// TIA Portal V20 export
TYPE "typeCmControlNodeInterlock"
// stored: Namespace Unit1.Em0
   STRUCT
      stacker1NgBoxLoading : "LER_typeTwoWayActuatorInterlock";
      stacker1NgBoxUnitMover : "LER_typeTwoWayActuatorInterlock";
      stacker1NgBoxClampLeft : "LER_typeTwoWayActuatorInterlock";
      stacker1NgBoxClampRight : "LER_typeTwoWayActuatorInterlock";
      stacker1NgBoxClampMover : "LER_typeTwoWayActuatorInterlock";
      stacker1NgBoxLift : "LER_typeTwoWayActuatorInterlock";
      stacker1NgBoxLock : "LER_typeTwoWayActuatorInterlock";
   END_STRUCT;
END_TYPE
